(* IEC 61131-3 sources: codesys-mcp-toolkit/standalone-sync/sources_st/511_05/DevLogic, 4 files *)

(* ---- FB_AutoHeater.fb.st ---- *)
// @OBJECT_ID: 0bcac0e8-eed9-4bae-8693-ddac31a98cce
// @DECLARATION
(*Рабочий алгоритм этого блока будет следующим: по переднему фронту сигнала xStart он включает внутренний пид-регулятор, который открывает клапан и начинает нагрев. Если xKeepTemp = FALSE, то как только текущая температура достигает заданной, мы снимаем сигнал разрешения (xEnable) и внутреннего пид-регулятора (нагрев прекращается). Если xKeepTemp = TRUE, то регулятор продолжает поддерживать температуру, пока активен xStart.
*)
FUNCTION_BLOCK FB_AutoHeater
VAR_INPUT
    xStart        : BOOL;   // Признак запуска нагрева (по переднему фронту)
    xKeepTemp     : BOOL;   // TRUE = поддерживать температуру после достижения, FALSE = отключить после нагрева (разовая операция)
    rTempActual   : REAL;   // Текущая температура в аппарате
    rTargetTemp   : REAL;   // Целевая температура, до которой нужно нагреть (или уставка)
    rTolerance    : REAL := 0.5; // Зона чувствительности (нагрев считается завершенным при Т >= уставка - Tolerance)
    // Параметры пид-регулятора
    rKp           : REAL := 1.0;
    rTn           : REAL := 10.0;
    rTv           : REAL := 0.0;
END_VAR
VAR_IN_OUT
    rValveOut     : REAL;   // Управляющее воздействие на клапан (0..100%)
    xAutoModeCmd  : BOOL;   // Выбор режима (TRUE = авто, FALSE = ручной)
END_VAR
VAR_OUTPUT
    xActive       : BOOL;   // Состояние: нагрев в процессе
    xDone         : BOOL;   // Состояние: нагрев успешно завершен (целевая Т достигнута)
END_VAR
VAR
    fbSteamControl : FB_UniversalSteamValveControl;
    xOldStart      : BOOL;  // Память сигнала запуска
    xEnablePID     : BOOL;  // Внутренний сигнал работы пид-регулятора
END_VAR

// @IMPLEMENTATION
// --- 1. Обработка команд и переходов состояний ---
// Детектор переднего фронта запуска: если пришел сигнал Start
IF xStart AND NOT xOldStart THEN
    xActive    := TRUE;   // Начинаем нагрев
    xDone      := FALSE;  // Сбрасываем флаг готовности
    xEnablePID := TRUE;   // Разрешаем работу внутреннего регулятора
END_IF;

// Условие достижения температуры
IF xActive AND (rTempActual >= (rTargetTemp - rTolerance)) THEN
    xDone := TRUE;   // Сигнализируем успешное достижение уставки

    // Если НЕ нужно удерживать температуру, выключаем нагрев
    IF NOT xKeepTemp THEN
        xActive    := FALSE;  // Останавливаем процесс
        xEnablePID := FALSE;  // Отключаем ПИД-регулятор
    END_IF;
END_IF;

// Обработка ручного сброса / выключения
IF NOT xStart THEN
    xDone := FALSE; // Сбрасываем статус при снятии Start
    IF xActive THEN
        xActive    := FALSE;
        xEnablePID := FALSE;
    END_IF;
END_IF;

xOldStart := xStart; // Запоминаем состояние фронта

// --- 2. Вызов регулирующего функционального блока ---
fbSteamControl(
    xEnable       := xEnablePID,
    rTempActual   := rTempActual,
    rSetpoint     := rTargetTemp,
    xReset        := FALSE,
    rKp           := rKp,
    rTn           := rTn,
    rTv           := rTv,
    rLimitLow     := 0.0,
    rLimitHigh    := 100.0,
    rValveOut     := rValveOut,
    xAutoModeCmd  := xAutoModeCmd
);

(* ---- FB_UniversalSteamValveControl.fb.st ---- *)
// @OBJECT_ID: c71aff23-84cd-4c4a-b310-a13f0d6eda39
// @DECLARATION
FUNCTION_BLOCK FB_UniversalSteamValveControl
VAR_INPUT
    xEnable       : BOOL;   // Переключатель контура (ВКЛ/ВЫКЛ) [1]
    rTempActual   : REAL;   // Текущая температура [1]
    rSetpoint     : REAL;   // Уставка температуры [1]
    xReset        : BOOL;   // Сброс ошибки ПИД [1]

    // Настройки ПИД (передаются снаружи для универсальности)
    rKp           : REAL;
    rTn           : REAL;
    rTv           : REAL;
    rLimitLow     : REAL;
    rLimitHigh    : REAL;
END_VAR

VAR_IN_OUT
    // Переменные IN_OUT изменяют внешнюю переменную по ссылке
    rValveOut     : REAL;   // Управляющее воздействие на клапан (0-100% или иное) [3]
    xAutoModeCmd  : BOOL;   // Команда режима: TRUE = АВТО, FALSE = РУЧНОЙ
END_VAR

VAR_OUTPUT
    xStatusActive : BOOL;   // Статус работы контура [1]
END_VAR

VAR
    fbPID         : oscat_basic.CTRL_PID; // Экземпляр ПИД из библиотеки Oscat [1]
    xOldEnable    : BOOL;   // Для детектора фронта [1]
    rInternalY    : REAL;   // Промежуточная переменная для выхода PID
END_VAR

// @IMPLEMENTATION

// --- ЛОГИКА ---

// 1. Управление режимами (детектирование изменения xEnable)
IF xEnable AND NOT xOldEnable THEN
    // ВКЛЮЧЕНИЕ:
    xStatusActive := TRUE;       // [2]
    xAutoModeCmd  := TRUE;       // Переводим внешний флаг в режим АВТО

ELSIF NOT xEnable AND xOldEnable THEN
    // ВЫКЛЮЧЕНИЕ:
    xStatusActive := FALSE;      // [2]
    xAutoModeCmd  := FALSE;      // Снимаем флаг АВТО (переход в ручной)
    rValveOut     := 0.0;        // Обнуляем выход на клапан [2]
END_IF;

xOldEnable := xEnable;

// 2. Вызов ПИД-регулятора
fbPID(
    ACT := rTempActual,          // [2]
    SET := rSetpoint,            // [2]
    MAN := NOT xStatusActive,    // Если не активен, ПИД в ручном режиме (MAN=TRUE) [2]
    RST := xReset,               // [2]
    KP  := rKp,                  // [2]
    TN  := MAX(rTn, 1.0),        // Защита от деления на 0, как в источнике [2]
    TV  := rTv,                  // [3]
    LL  := rLimitLow,            // [3]
    LH  := rLimitHigh            // [3]
);

// 3. Передача значения из ПИД во внешнюю переменную через IN_OUT
// Обновляем выход только если контур активен, чтобы не перебивать ручное управление при выключенном блоке
IF xStatusActive THEN
    rValveOut := fbPID.Y;        // [3]
END_IF;

(* ---- FB_ValveS_Compact.fb.st ---- *)
// @OBJECT_ID: fa77258a-480d-4f24-958d-df1ed5a50eb2
// @DECLARATION
FUNCTION_BLOCK FB_ValveS_Compact
VAR_INPUT
    xMode        : BOOL;
    xManControl  : BOOL;
    xAutoControl : BOOL;
END_VAR

VAR_OUTPUT
    xOutControl  : BOOL;
END_VAR

// @IMPLEMENTATION
// Компактная реализация в одну строку с помощью SEL
xOutControl := SEL(xMode, xManControl, xAutoControl);

(* ---- fbElemerREM.fb.st ---- *)
// @OBJECT_ID: f24ff6c8-e667-4d1a-8a4a-3707ce6a677c
// @DECLARATION
(* ИСПРАВЛЕНИЕ v4.1.0:
        - Исправлен разбор lrTotalVolume (LREAL / Double 64 бит).
        - Прибор передаёт регистры в порядке Big-Endian (src[0] = MSW, src[3] = LSW).
        - ЦПУ ПЛК — Little-Endian, поэтому выполняется разворот по WORD-словам:
          pW[3] = src[0] (старший), pW[0] = src[3] (младший).
        - Побайтовый подход заменён на пословный (POINTER TO WORD) — корректнее
          и безопаснее, так как каждый WORD внутри уже находится в правильном
          байтовом порядке аппаратуры Little-Endian.
*)

FUNCTION_BLOCK fbElemerREM
VAR_INPUT
    pFlowBuffer         : POINTER TO ARRAY[0..1] OF WORD;  (* Канал 0: Мгновенный расход F2, 2 регистра WORD *)
    pVolumeBuffer       : POINTER TO ARRAY[0..3] OF WORD;  (* Канал 1: Накопленный объём F1, 4 регистра WORD *)
    xCommError          : BOOL;                             (* Признак ошибки связи (из статуса Modbus Slave) *)
    xEnableLog          : BOOL := TRUE;                     (* Флаг разрешения детального логирования на HMI *)
END_VAR
VAR_IN_OUT
    xResetTotalizer     : BOOL;  (* Команда сброса сумматора с HMI — автосброс после выполнения *)
END_VAR
VAR_OUTPUT
    xDataValid          : BOOL;         (* Флаг достоверности данных для контуров ТАУ *)
    rInstantFlow        : REAL;         (* Мгновенный расход F2, куб.м/ч *)
    lrTotalVolume       : LREAL;        (* Накопленный общий объём F1, куб.м *)
    sStatus             : STRING(255);  (* Строка текущего шага для оператора панели *)
END_VAR
VAR
    (* Автомат состояний *)
    eState              : E_REM_State;
    eLastState          : E_REM_State;

    (* Указатели для разбора REAL (32 бит) *)
    pByteSrc            : POINTER TO BYTE;
    pByteDst            : POINTER TO BYTE;
    dwRealParser        : DWORD;

    (* Указатель для разбора LREAL (64 бит) — пословный разворот *)
    pWordDst            : POINTER TO WORD;  (* Указатель на LREAL как массив из 4 WORD *)

    (* Системные таймеры *)
    tonStateTimer       : TON;
    udiMinutesInState   : UDINT;
END_VAR
VAR CONSTANT
    DEVICE_DISCONNECTED : REAL := -10000.0;  (* Маркер аварии датчика *)
END_VAR

// @IMPLEMENTATION
//==============================================================================
// Расчёт времени нахождения в текущем состоянии (в минутах для HMI)
//==============================================================================
tonStateTimer(IN := (eState = eLastState), PT := T#240h);
udiMinutesInState := TIME_TO_UDINT(tonStateTimer.ET) / 60000;

//==============================================================================
// 1. ДИАГНОСТИЧЕСКИЙ КОНТРОЛЬ АВАРИЙ СВЯЗИ ВЕРХНЕГО УРОВНЯ
//==============================================================================
IF xCommError THEN
    eState := E_REM_State.ERROR_COMM;
ELSIF xResetTotalizer AND eState <> E_REM_State.ERROR_COMM THEN
    eState := E_REM_State.RESET_LOGIC;
ELSIF eState <> E_REM_State.ERROR_COMM AND eState <> E_REM_State.RESET_LOGIC THEN
    eState := E_REM_State.OPERATING;
END_IF;

//==============================================================================
// 2. СТРУКТУРА СТЕЙТ-МАШИНЫ
//==============================================================================
CASE eState OF

    E_REM_State.INIT: //--------------------------------------------------------
        sStatus        := 'ЭЛЕМЕР-РЭМ: Ожидание первого скана и данных от Modbus-каналов';
        rInstantFlow   := DEVICE_DISCONNECTED;
        lrTotalVolume  := LREAL#-10000.0;
        xDataValid     := FALSE;

        IF pFlowBuffer <> 0 AND pVolumeBuffer <> 0 AND NOT xCommError THEN
            eState := E_REM_State.OPERATING;
        END_IF;

    E_REM_State.OPERATING: //---------------------------------------------------
        sStatus := 'ЭЛЕМЕР-РЭМ: Данные успешно обновляются, идёт технологический учёт';

        IF pFlowBuffer <> 0 AND pVolumeBuffer <> 0 THEN

            // ----------------------------------------------------------------
            // РАЗБОР МГНОВЕННОГО РАСХОДА F2
            // Канал 0, REAL 32 бита, формат прибора DCBA (Big-Endian)
            // Побайтовый разворот → Little-Endian ЦПУ ПЛК
            // ----------------------------------------------------------------
            pByteSrc := ADR(pFlowBuffer^[0]);
            pByteDst := ADR(dwRealParser);

            IF pByteSrc <> 0 AND pByteDst <> 0 THEN
                pByteDst[0] := pByteSrc[3]; // D → LSB
                pByteDst[1] := pByteSrc[2]; // C
                pByteDst[2] := pByteSrc[1]; // B
                pByteDst[3] := pByteSrc[0]; // A → MSB
                SysMemCpy(pDest := ADR(rInstantFlow), pSrc := ADR(dwRealParser), udiCount := SIZEOF(rInstantFlow));
            END_IF;

            // ----------------------------------------------------------------
            // РАЗБОР НАКОПЛЕННОГО ОБЪЁМА F1
            // Канал 1, Double/LREAL 64 бита, Big-Endian порядок WORD-регистров:
            //   src[0] = MSW (старший), src[3] = LSW (младший)
            //
            // Алгоритм прибора (из документации):
            //   v  = (uint64_t)src[0] << 48
            //   v |= (uint64_t)src[1] << 32
            //   v |= (uint64_t)src[2] << 16
            //   v |= (uint64_t)src[3]
            //
            // На Little-Endian ЦПУ ПЛК LREAL в памяти хранится так:
            //   pW[0] = LSW (биты  0..15)
            //   pW[1]        (биты 16..31)
            //   pW[2]        (биты 32..47)
            //   pW[3] = MSW (биты 48..63)
            //
            // Поэтому разворачиваем порядок WORD-ов:
            //   pW[3] := src[0]   (MSW прибора → старший WORD LREAL)
            //   pW[2] := src[1]
            //   pW[1] := src[2]
            //   pW[0] := src[3]   (LSW прибора → младший WORD LREAL)
            //
            // Байты ВНУТРИ каждого WORD НЕ трогаем — аппаратура ПЛК
            // уже прочитала их корректно в Little-Endian.
            // ----------------------------------------------------------------
            pWordDst := ADR(lrTotalVolume);

            IF pWordDst <> 0 THEN
                pWordDst[3] := pVolumeBuffer^[0]; // MSW прибора → старший WORD
                pWordDst[2] := pVolumeBuffer^[1];
                pWordDst[1] := pVolumeBuffer^[2];
                pWordDst[0] := pVolumeBuffer^[3]; // LSW прибора → младший WORD
            END_IF;

            // ----------------------------------------------------------------
            // ЗАЩИТА ТАУ: Валидация на NaN
            // ----------------------------------------------------------------
            IF rInstantFlow <> rInstantFlow OR lrTotalVolume <> lrTotalVolume THEN
                sStatus    := 'ЭЛЕМЕР-РЭМ: Критическая ошибка! Считано неопределённое значение NaN.';
                xDataValid := FALSE;
            ELSE
                xDataValid := TRUE;
            END_IF;

        ELSE
            sStatus    := 'ЭЛЕМЕР-РЭМ: Внимание, обнаружен нулевой указатель буферов опроса!';
            xDataValid := FALSE;
        END_IF;

    E_REM_State.RESET_LOGIC: //-------------------------------------------------
        sStatus    := 'ЭЛЕМЕР-РЭМ: Выполняется процедура сброса сумматора по команде оператора';
        xDataValid := TRUE;

        IF NOT xResetTotalizer THEN
            eState := E_REM_State.OPERATING;
        END_IF;

    E_REM_State.ERROR_COMM: //--------------------------------------------------
        sStatus       := 'АВАРИЯ связи: Прибор не отвечает. Проверьте кабель RS-485!';
        rInstantFlow  := DEVICE_DISCONNECTED;
        lrTotalVolume := LREAL#-10000.0;
        xDataValid    := FALSE;

        IF NOT xCommError THEN
            eState := E_REM_State.INIT;
        END_IF;

END_CASE;

//==============================================================================
// 3. ДИАГНОСТИЧЕСКОЕ ЛОГИРОВАНИЕ ДЛЯ ОПЕРАТОРА ПАНЕЛИ
//==============================================================================
IF xEnableLog AND (eState <> eLastState) THEN
    eLastState := eState;
    sStatus    := CONCAT(sStatus, CONCAT(' | Прошло времени: ', UDINT_TO_STRING(udiMinutesInState)));
    sStatus    := CONCAT(sStatus, ' мин.');
END_IF;
